// TIA Portal V17 export
// export: Created 2025-04-11T04:54:23.8909083Z, ExportSetting WithDefaults, DisplayName Totally Integrated Automation Portal, DisplayVersion V17, DisplayName TIA Portal Openness, DisplayVersion V17, DisplayName TIA Portal Version Control Interface, DisplayVersion V17, DisplayName SINAMICS Startdrive Advanced, DisplayVersion V17, DisplayName SINAMICS Startdrive G130, G150, S120, S150, SINAMICS MV, S210, DisplayVersion V17, DisplayName SINAMICS Startdrive G110M, G120, G120C, G120D, G120P, G115D, DisplayVersion V17, DisplayName STEP 7 Professional, DisplayVersion V17, DisplayName STEP 7 Safety, DisplayVersion V17, DisplayName WinCC Advanced, DisplayVersion V17
TYPE "UDT_Device_Temp"
// stored: IsFailsafeCompliant false
   STRUCT
      IN_xAutoCmd : Bool;   // 自动模式启动设备
      IN_xManualCmd : Bool;   // 手动模式下的设备控制辅助命令/1为启动，0为停止
      IN_xStartCondition : Bool := TRUE;   // 启动设备运行条件
      OUT_xStartOK : Bool;   // 启动到位
      OUT_xStopOK : Bool;   // 停止到位
   END_STRUCT;
END_TYPE
